(* PLC project Beremiz non-standard POUs library, LOLITECH Beremiz 0.0 *)
(* stored: creationDateTime 2008-12-14T16:53:26, modificationDateTime 2008-12-23T22:35:46 *)

FUNCTION_BLOCK python_eval
  VAR_INPUT
    TRIG : BOOL;
    CODE : STRING;
  END_VAR
  VAR_OUTPUT
    ACK : BOOL;
    RESULT : STRING;
  END_VAR
  VAR
    STATE : DWORD;
    BUFFER : STRING;
    PREBUFFER : STRING;
    TRIGM1 : BOOL;
    TRIGGED : BOOL;
  END_VAR

{extern void __PythonEvalFB(int, PYTHON_EVAL*);__PythonEvalFB(0, data__);}
          
END_FUNCTION_BLOCK

FUNCTION_BLOCK python_poll
  VAR_INPUT
    TRIG : BOOL;
    CODE : STRING;
  END_VAR
  VAR_OUTPUT
    ACK : BOOL;
    RESULT : STRING;
  END_VAR
  VAR
    STATE : DWORD;
    BUFFER : STRING;
    PREBUFFER : STRING;
    TRIGM1 : BOOL;
    TRIGGED : BOOL;
  END_VAR

{extern void __PythonEvalFB(int, PYTHON_EVAL*);__PythonEvalFB(1,(PYTHON_EVAL*)(void*)data__);}
          
END_FUNCTION_BLOCK
